Staubli VAL3: load.pgx

public program load(string x_sItem (dimensions=1), num& x_nResult (dimensions=1))
  local num i
  local string l_sMessage
  local string l_sType
begin
  // load the select trajectory..already loaded
  call getTrajType(l_sType)
  if find(pt:libPath(),saveData:sPathTraj)==-1
    pt:libLoad(saveData:sPathTraj+l_sType)
    delay(0)
    if saveData:bDebug
      ? "loading TRAJ..."+saveData:sPathTraj+l_sType
    endIf
  endIf
  // use the type...
  if isDefined(pt:tTraj[x_sItem])
    // link the frame and all the points
    call pt:link_all(x_sItem)
    // check if link and defined
    pEditPoint=pt:tTraj[x_sItem]
    // link all
    link(pEditPoint.fFrame,world)
    for i=0 to size(pEditPoint.tData)-1
      link(pEditPoint.tData[i].pPoint,pEditPoint.fFrame)
      link(pEditPoint.tData[i].pCircle,pEditPoint.fFrame)
    endFor
    pEditPoint.sID=x_sItem
  elseIf x_sItem!=""
    // not FOUND
    call language:message(l_sMessage,-7)
    x_nResult=-1
    popUpMsg(l_sMessage+x_sItem)
  endIf
end
